(*
Provides methods and properties to operate on RGBA value.
*)
FUNCTION_BLOCK Argbb IMPLEMENTS I_Argbb
VAR
	_r: BYTE;
	_g: BYTE;
	_b: BYTE;
	_a: BYTE;
END_VAR

(*
ALPHA channel
*)
PROPERTY Alpha : BYTE
GET
Alpha := _a;
END_GET
SET
_a := Alpha;
END_SET
END_PROPERTY

(*
BLUE component
*)
PROPERTY Blue : BYTE
GET
Blue := _b;
END_GET
SET
_b := Blue;
END_SET
END_PROPERTY

(*
Clones other components of I_RgbaColor interface.
*)
METHOD Clone
VAR_INPUT
	iColor	: I_Argbb;
END_VAR
IF iColor = 0 THEN
	RETURN;
END_IF

_r := iColor.Red;
_b := iColor.Blue;
_g := iColor.Green;
_a := iColor.Alpha;
END_METHOD

{attribute 'hide'}
METHOD FB_init : BOOL
VAR_INPUT
	bInitRetains : BOOL;
	bInCopyCode : BOOL;
	nRed: USINT;
	nGreen: USINT;
	nBlue: USINT;
	nAlpha: USINT;
END_VAR
Set(nRed, nGreen, nBlue, nAlpha);
END_METHOD

(*
GREEN component
*)
PROPERTY Green : BYTE
GET
Green := _g;
END_GET
SET
_g := Green;
END_SET
END_PROPERTY

(*
Compute single Color value from RGBA components when used as getter.
Sets RGBA values by extracting components from a single Color value.
*)
PROPERTY Raw : Argb
GET
Raw := 	USINT_TO_UDINT(_b) OR
			SHL(USINT_TO_UDINT(_g), 8) OR
			SHL(USINT_TO_UDINT(_r), 16) OR
			SHL(USINT_TO_UDINT(_a), 24);
END_GET
SET
_b := UDINT_TO_USINT(Raw AND 16#FF);
_g := UDINT_TO_USINT(SHR(Raw, 8) AND 16#FF);
_r := UDINT_TO_USINT(SHR(Raw, 16) AND 16#FF);
_a := UDINT_TO_USINT(SHR(Raw, 24) AND 16#FF);
END_SET
END_PROPERTY

(*
RED component
*)
PROPERTY Red : BYTE
GET
Red := _r;
END_GET
SET
_r := Red;
END_SET
END_PROPERTY

(*
Set each RGBA component value separately.
*)
METHOD Set
VAR_INPUT
	nRed: USINT;
	nGreen: USINT;
	nBlue: USINT;
	nAlpha: USINT;
END_VAR
_r := nRed;
_g := nGreen;
_b := nBlue;
_a := nAlpha;
END_METHOD

END_FUNCTION_BLOCK

(* stored: Version 1.1.0.1
   POU Argbb: Id {2722e4a4-8a93-411e-a3ea-39a44af2a9e8}, SpecialFunc None
   Property Alpha: Id {61fe6c55-bd71-4e71-af28-24097f508d00}
   Get Get: Id {9d4821de-72dd-444c-991c-d2ec0cdd3814}
   Set Set: Id {f95f74b8-ca7b-4373-af0d-46fdb9bbbf45}
   Property Blue: Id {0473fd13-3e4a-46cd-92d1-78e19c1e7bc2}
   Get Get: Id {8570242d-e6c6-4d02-a710-93e6cf52eda1}
   Set Set: Id {7d59663d-3256-4403-9f6d-a0789082fe6f}
   Method Clone: Id {924c2e5f-fff2-4c25-9bf1-439819cf4eda}
   Method FB_init: Id {8f277162-e746-4b57-9ebb-b150327f2243}
   Property Green: Id {8ec01b6b-1c45-4d2c-91da-d78954155238}
   Get Get: Id {41b4783c-4227-4b80-93ac-7e4b95b6953a}
   Set Set: Id {5aa334fc-967a-4a58-9f0e-1b62e94feb7c}
   Property Raw: Id {2c7b24d8-afcd-4243-8d9f-839ca3e0e22f}
   Get Get: Id {101e36a2-7284-4e50-b5a7-31e84ab6f554}
   Set Set: Id {533060d0-5fac-4157-9799-d508600c2958}
   Property Red: Id {cec73e8f-0e69-462b-8b4d-1f0aa08c453e}
   Get Get: Id {eceb49b4-def0-4258-8e6c-43d57dab2ccf}
   Set Set: Id {c443a33b-699f-4236-a822-e87eea3966eb}
   Method Set: Id {1d8ceed2-bd8a-4471-aa42-fc7ee85534e9} *)
